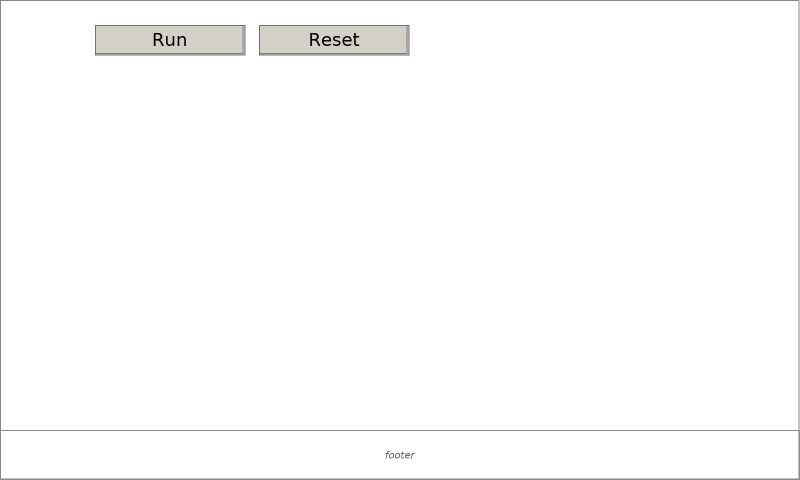
VISUALIZATION Visualization  // 800x480
    Button (95,25 150x30), "Run"
        toggle G_Safety.runSafety
    Button (259,25 150x30), "Reset"
        tap G_Safety.resetSafety
    Frame (0,430 800x50)
        shows footer()
END_VISUALIZATION

(* stored: Version 1.1.0.1, ProductVersion 3.1.4024.12
   Visu Visualization: Id {1ef672dd-8b31-492d-80a3-c62b95812e19} *)
